// TIA Portal V16 export
// export: Created 2025-05-30T16:36:00.0343468Z, ExportSetting WithDefaults, DisplayName Totally Integrated Automation Portal, DisplayVersion V16, DisplayName TIA Portal Version Control Interface, DisplayVersion V16, DisplayName TIA Portal Openness, DisplayVersion V16, DisplayName STEP 7 Professional, DisplayVersion V16, DisplayName STEP 7 Safety, DisplayVersion V16, DisplayName WinCC Advanced, DisplayVersion V16
FUNCTION_BLOCK "FB_EncoderFeedback_Degree"   // FB19, FBD
VERSION : 0.1
// stored: AutoNumber true, IsIECCheckEnabled false, UDAEnableTagReadback false
   VAR_INPUT
      CounterTag { ExternalVisible := 'False'; ExternalWritable := 'False'} : Int;   // Connect to the CounterTag IW102
      Position_Offset { ExternalVisible := 'False'; ExternalWritable := 'False'} : Real;   // Fill in the tolerance, when the axis approves the position. Above or below the desired position
      Pulsfactor { ExternalVisible := 'False'; ExternalWritable := 'False'} : Real;   // Number of pulses after 360 degree turn of the axis.
      Position_Correction { ExternalVisible := 'False'; ExternalWritable := 'False'} : Real;   // Small Position Correction for the Axis
      ReferenceRun_Command { ExternalVisible := 'False'; ExternalWritable := 'False'} : Bool;   // Command of starting the referencerun
      ReferenceSwitch { ExternalVisible := 'False'; ExternalWritable := 'False'} : Bool;   // ReferenceSwitch Mounted on Axis
      ReferencePosition { ExternalVisible := 'False'; ExternalWritable := 'False'} : Int;   // Position where the index puls of the reference switch enters.
   END_VAR
   VAR_OUTPUT
      Scaled_Position { ExternalVisible := 'False'; ExternalWritable := 'False'} : Real;   // Scaled Position scaled with Pulsfactor
      Actual_Enc_Pos { ExternalVisible := 'False'; ExternalWritable := 'False'} : Real;   // Actual Encoder Position
      AxisDB_Connection { ExternalVisible := 'False'; ExternalWritable := 'False'} : Real;   // Connection with Axis DB connection
   END_VAR
   VAR_TEMP
      Corrected_Axis_Pos : Real;
      Unscaled_Position : Int;   // Unscaled Position of the Encoder
      Unsc2 : Int;   // Unsc 2 position
      Act_Enc_Pos_Int : DInt;
      Scaled_Position_Real : Real;
      PosDint : DInt;
      Unscaled_Position_Real : Real;
      InternalCounter : Int;
      CalDifCounter : Int;
      Pos_Storage : Int;
      Pos_Diffrence : Int;
      Add_Pos : Int;
      Sub_Pos : Int;
      LessThanZero : Bool;
      LTZ_out : Int;
   END_VAR
BEGIN

REGION Network 2: SPARE
END_REGION

NETWORK
TITLE = Call the Countermodule
      L     #CounterTag;  //Van tellerkaart TAG Gelinkt aan IW102
      L     "PositionManagement".Data.CntPlsPrev;  //Vorige scan
      -D;
      T     "PositionManagement".Data.CntPlsDiff;  //Verschil

      L     "PositionManagement".Data.CntPlsDiff;  // Verschil groter dan nul?
      L     0;
      >D;
      JCN   chkneg;

      L     "PositionManagement".Data.CntPlsDiff;  //Verschil optellen bij actuele pulswaarde
      L     "PositionManagement".Data.CntPlsAct;
      +D;
      T     "PositionManagement".Data.CntPlsAct;
      JU    end;  //rest overslaan.

chkneg:L     "PositionManagement".Data.CntPlsDiff;  // Verschil groter dan nul?
      L     0;
      <D;
      JCN   end;
      L     -1;  //verschil positief maken
      *D;
      T     "PositionManagement".Data.CntPlsDiff;  //verschil positief

      L     "PositionManagement".Data.CntPlsAct;  //Verschil optellen bij actuele pulswaarde
      +D;
      T     "PositionManagement".Data.CntPlsAct;

end:  NOP   0;

      L     #CounterTag;
      T     "PositionManagement".Data.CntPlsPrev;


REGION Network 4: Store Old Position
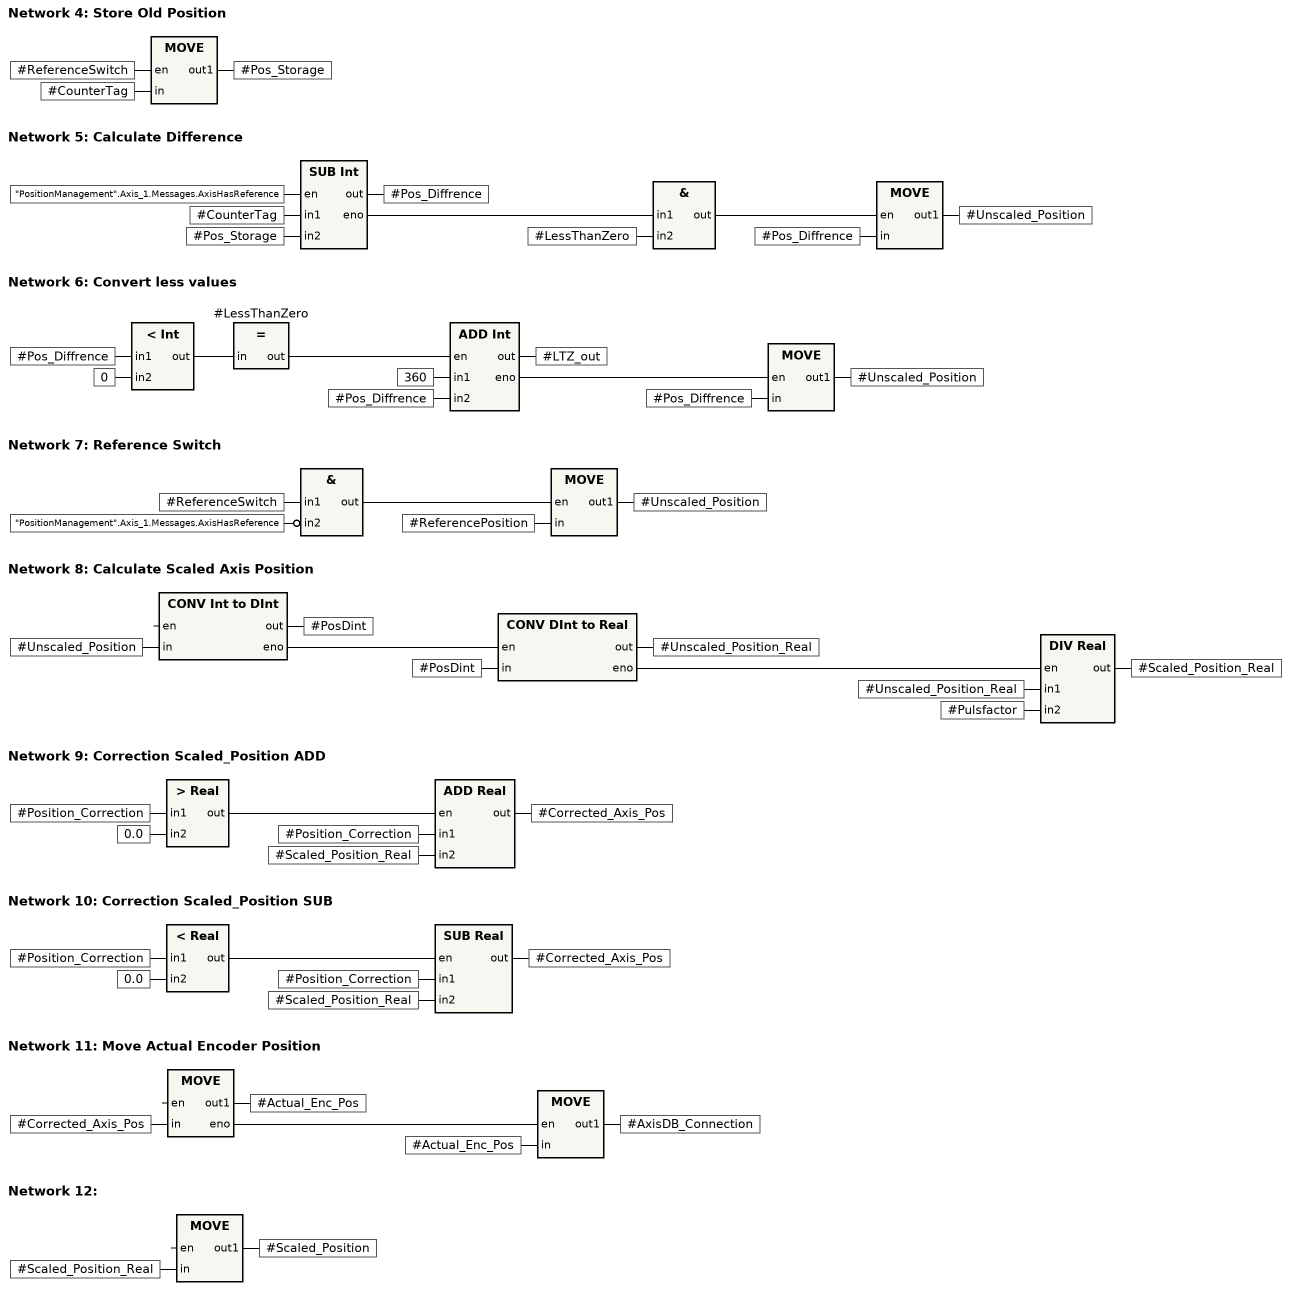
   IF #ReferenceSwitch THEN #Pos_Storage := #CounterTag; END_IF;
END_REGION

REGION Network 5: Calculate Difference
   // ENO of a box is taken as its EN; it also drops when the box reports an error
   IF "PositionManagement".Axis_1.Messages.AxisHasReference THEN
       #Pos_Diffrence := #CounterTag - #Pos_Storage;
   END_IF;
   IF "PositionManagement".Axis_1.Messages.AxisHasReference AND #LessThanZero THEN
       #Unscaled_Position := #Pos_Diffrence;
   END_IF;
END_REGION

REGION Network 6: Convert less values
   // ENO of a box is taken as its EN; it also drops when the box reports an error
   #LessThanZero := #Pos_Diffrence < 0;
   IF #LessThanZero THEN
       #LTZ_out := 360 + #Pos_Diffrence;
       #Unscaled_Position := #Pos_Diffrence;
   END_IF;
END_REGION

REGION Network 7: Reference Switch
   IF #ReferenceSwitch AND NOT "PositionManagement".Axis_1.Messages.AxisHasReference THEN
       #Unscaled_Position := #ReferencePosition;
   END_IF;
END_REGION

REGION Network 8: Calculate Scaled Axis Position
   // ENO of a box is taken as its EN; it also drops when the box reports an error
   #PosDint := INT_TO_DINT(#Unscaled_Position);
   #Unscaled_Position_Real := DINT_TO_REAL(#PosDint);
   #Scaled_Position_Real := #Unscaled_Position_Real / #Pulsfactor;
END_REGION

REGION Network 9: Correction Scaled_Position ADD
   IF #Position_Correction > 0.0 THEN
       #Corrected_Axis_Pos := #Position_Correction + #Scaled_Position_Real;
   END_IF;
END_REGION

REGION Network 10: Correction Scaled_Position SUB
   IF #Position_Correction < 0.0 THEN
       #Corrected_Axis_Pos := #Position_Correction - #Scaled_Position_Real;
   END_IF;
END_REGION

REGION Network 11: Move Actual Encoder Position
   // ENO of a box is taken as its EN; it also drops when the box reports an error
   #Actual_Enc_Pos := #Corrected_Axis_Pos;
   #AxisDB_Connection := #Actual_Enc_Pos;
END_REGION

REGION Network 12
   #Scaled_Position := #Scaled_Position_Real;
END_REGION
END_FUNCTION_BLOCK
